// TIA Portal V20 export
TYPE "zp_CITICoS"
// stored: Access Published, Namespace CITI_Logic
   STRUCT
      Map_ID : SInt;
      Material_Low_Warning : Bool;
      Auto_Cycle_Running : Bool;
      Manual_Mode : Bool;
      Cycle_Time_Ready : Bool;
      Overcycle : Bool;
      OperatorOvercycle1 : Bool;
      OperatorOvercycle2 : Bool;
      Blocked : Bool;
      Starved : Bool;
      Idle : Bool;
      Wait_1 : Bool;
      Wait_2 : Bool;
      Wait_3 : Bool;
      Wait_4 : Bool;
      Stopped_by_Operator : Bool;
      Machine_Fault : Bool;
      Machine_Fault_Ack : Bool;
      Quality_Check_Warning : Bool;
      Quality_Check_Fault : Bool;
      Quality_Check_Ack : Bool;
      Tool_Change_Warning : Bool;
      Tool_Change_Fault : Bool;
      Tool_Change_Ack : Bool;
      Spare_Bool_1 : Bool;
      Station_Andon_Hold : Bool;
      Filter_Minor_Fault : Bool;
      Filter_Tank_Coolant_Temp_OK : Bool;
      Filter_Tank_Coolant_Temp_High : Bool;
      Filter_Tank_Coolant_Temp_Low : Bool;
      Filter_Tank_Level_OK : Bool;
      Filter_Tank_Level_High : Bool;
      Filter_Tank_Level_Low : Bool;
      Filter_PumpBack_Level_OK : Bool;
      Filter_PumpBack_Level_High : Bool;
      Filter_PumpBack_Level_Low : Bool;
      CMM_Bad_Quality_Data_Available : Bool;
      CMM_No_Que_Available : Bool;
      CMM_Que_Available : Bool;
      CMM_Inspection_Program_Running : Bool;
      Spare_Bool_2 : Bool;
      CMM_Program_Minutes_Remaining : Int;
      Date_of_Event : DInt;
      Time_of_Event : DInt;
      Fault_Word : DInt;
   END_STRUCT;
END_TYPE
